{attribute 'reflection'}
FUNCTION_BLOCK ABSTRACT FB_BaseFB IMPLEMENTS I_BaseFB
VAR
  {attribute 'instance-path'}
  {attribute 'noinit'}
  InstancePath : STRING;
END_VAR

// I_BaseFB
VAR
  _Busy : BOOL := TRUE;
  _Error : BOOL;
  _ErrorID : UDINT;
END_VAR

// Derivatives of FB_BaseFB can have code in the function block body

PROPERTY Busy : BOOL
GET
Busy := _Busy;
END_GET
END_PROPERTY

PROPERTY Error : BOOL
GET
Error := _Error;
END_GET
END_PROPERTY

PROPERTY ErrorID : UDINT
GET
ErrorID := _ErrorID;
END_GET
END_PROPERTY

METHOD PUBLIC Marker
VAR_INPUT
  Message : T_MaxString;
END_VAR
Tracing.GlobalTraceLog.AddEntry(InstancePath, Message, 1);
END_METHOD

METHOD PUBLIC Trace
VAR_INPUT
  Message : T_MaxString;
END_VAR
Tracing.GlobalTraceLog.AddEntry(InstancePath, Message, 0);
END_METHOD

METHOD PUBLIC TraceWithJson
VAR_INPUT
  Message : T_MaxString;
  Json : T_MaxString;
END_VAR
Tracing.GlobalTraceLog.AddEntryWithJson(
  InstancePath,
  Message,
  0,
  Json
);
END_METHOD

END_FUNCTION_BLOCK

(* stored: Version 1.1.0.1, ProductVersion 3.1.4024.12
   POU FB_BaseFB: Id {6ed07efa-981d-468f-96e4-311962a2c1b8}, SpecialFunc None
   Folder I_BaseFB: Id {2446e10f-9689-4d09-8275-cafb17936ff6}
   Property Busy: Id {4d6cbdf9-39d1-402a-bdf7-e99c763ca664}
   Get Get: Id {510bfdb9-9653-47e3-8858-155884e2d528}
   Property Error: Id {34ee3fc8-e733-4c8d-957d-73debe23ad7c}
   Get Get: Id {b329f8a8-e324-48ec-9892-094f3f1b91ee}
   Property ErrorID: Id {7222581b-9e78-401f-a0dd-949f1d909b6b}
   Get Get: Id {733202ff-38c2-4e4c-bf03-c44f4b2507c6}
   Method Marker: Id {3f6d42cb-413f-01fd-1c14-04724641b65a}
   Method Trace: Id {eba63575-88fd-04fd-3b9f-7fd7e52b185c}
   Method TraceWithJson: Id {2f3817ed-644b-49e3-896f-ee1fa4905779} *)
